# EPICS alarm handler configuration: mps_database/bare/alarms/areas/mpln_undh_mp05.alhConfig
GROUP NULL MPLN:UNDH:MP05:1
$ALIAS MPS Link Node 140
$GUIDANCE
LTUH MPS
   Group Name: MPLN:UNDH:MP05:1
   Summary PV:  MPLN:UNDH:MP05:1:STATSUMY
$END
CHANNEL  MPLN:UNDH:MP05:1    MPLN:UNDH:MP05:1:MPS_EN_RBV		-----
CHANNEL  MPLN:UNDH:MP05:1    MPLN:UNDH:MP05:1:LC1_MODE_RBV		-----
